FUNCTION ASCF_CL_34_NOR : WORD
VAR_OUTPUT
	Out						: ASCF_UnionType;		//Result of the computation (Type: VBool or VDWord)
END_VAR

VAR_IN_OUT
	Arguments				: ARRAY[0..3] OF ASCF_UnionType;	//Arguments for the function (Arguments: 2 - 4, Type: VBool or VDWord)
END_VAR

VAR
	tempRet					: WORD;
	constErrors				: ASCF_CL_EnumErrors;				//Enumeration type of the error codes of the Adaptive Logic.
END_VAR



//#################################################################################################
{region "EXECUTE AND OUTPUT"}
    tempRet := ASCF_CL_32_OR(Arguments := Arguments, Out => Out);
    
    // negate result if OR was successful
    IF tempRet = constErrors.None THEN
        Out.VBool := NOT Out.VBool;
    END_IF;
    
    ASCF_CL_34_NOR := tempRet;
{endregion}

END_FUNCTION

(* stored: Version 1.1.0.1, ProductVersion 3.1.4026.4
   POU ASCF_CL_34_NOR: Id {cab1610f-d5c2-497e-a5e9-f33b202b2db8}, SpecialFunc None *)
